// TIA Portal V17 export
// export: Created 2022-07-20T07:01:33.8166231Z, ExportSetting WithDefaults, DisplayName Totally Integrated Automation Portal, DisplayVersion V17, DisplayName TIA Portal Openness, DisplayVersion V17, DisplayName TIA Portal Version Control Interface, DisplayVersion V17, DisplayName SINAMICS Startdrive Advanced, DisplayVersion V17, DisplayName SINAMICS Startdrive G130, G150, S120, S150, SINAMICS MV, S210, DisplayVersion V17, DisplayName SINAMICS Startdrive G110M, G120, G120C, G120D, G120P, G115D, DisplayVersion V17, DisplayName STEP 7 Professional, DisplayVersion V17, DisplayName STEP 7 Safety, DisplayVersion V17, DisplayName WinCC Advanced, DisplayVersion V17
FUNCTION_BLOCK "FB10323_PrinterCompactAirCircuit"   // FB10323, LAD
{ S7_Optimized_Access := 'TRUE' }
VERSION : 0.1
// stored: AutoNumber false, IsIECCheckEnabled false, IsRetainMemResEnabled false, MemoryReserve 100, SetENOAutomatically false, UDAEnableTagReadback false
   VAR_INPUT
      AirCircuit_MainVacuum_VacuumSensor_raw : Int;
      AirCircuit_B1_VacuumSensor_raw : Int;
      AirCircuit_B2_VacuumSensor_raw : Int;
      AirCircuit_MainVacuum_Setpoint_mbar : Real;
      AirCircuit_B1_Setpoint_mbar : Real;
      AirCircuit_B2_Setpoint_mbar : Real;
      AirCircuitParameterB1PurgeTime_s : Time;
      AirCircuitParameterB2PurgeTime_s : Time;
   END_VAR
   VAR_OUTPUT
      AirCircuit_MainVacuum_SolenoidValve : Bool;
      AirCircuit_MainVacuum_Pump : Bool;
      AirCircuit_B1_JunctionMainVaccum_SolenoidValve : Bool;
      AirCircuit_B1_Tank_SolenoidValve : Bool;
      AirCircuit_B1_Venting_SolenoidValve : Bool;
      AirCircuit_B1_Purge_SolenoidValve : Bool;
      AirCircuit_B1_Purge_Pump : Bool;
      AirCircuit_B1_PurgeDone : Bool;
      AirCircuit_B2_JunctionMainVaccum_SolenoidValve : Bool;
      AirCircuit_B2_Tank_SolenoidValve : Bool;
      AirCircuit_B2_Venting_SolenoidValve : Bool;
      AirCircuit_B2_Purge_SolenoidValve : Bool;
      AirCircuit_B2_Purge_Pump : Bool;
      AirCircuit_B2_PurgeDone : Bool;
      EnablePWM : Bool;
      PumpDutyCycle : Int;
      MainVacuumActualValue : Real;
      B1VacuumActualValue : Real;
      AutoRegulationB1Done : Bool;
      B2VacuumActualValue : Real;
      AutoRegulationB2Done : Bool;
      AutoRegulationB1_B2_Done : Bool;
   END_VAR
   VAR_IN_OUT
      AirCircuitRequestAutoregulation : Bool;
      AirCircuitRequestMainVacuumRegulation : Bool;
      AirCircuitRequestB1Regulation : Bool;
      AirCircuitRequestB2Regulation : Bool;
      AirCircuitRequestB1Purge : Bool;
      AirCircuitRequestB2Purge : Bool;
   END_VAR
   VAR
      MainVacuumStateDiagram : Int;
      B1VacuumStateDiagram : Int;
      B2VacuumStateDiagram : Int;
      R_TRIG_RequestAutoregulationAirCircuit : R_TRIG;
      F_TRIG_RequestAutoregulationAirCircuit { S7_SetPoint := 'True'} : F_TRIG;
      R_TRIG_RequestMainVacuumRegulation { S7_SetPoint := 'True'} : R_TRIG;
      F_TRIG_RequestMainVacuumRegulation { S7_SetPoint := 'True'} : F_TRIG;
      R_TRIG_RequestB1Regulation { S7_SetPoint := 'True'} : R_TRIG;
      F_TRIG_RequestB1Regulation { S7_SetPoint := 'True'} : F_TRIG;
      R_TRIG_RequestB2Regulation { S7_SetPoint := 'True'} : R_TRIG;
      F_TRIG_RequestB2Regulation { S7_SetPoint := 'True'} : F_TRIG;
      R_TRIG_RequestB1Purge { S7_SetPoint := 'True'} : R_TRIG;
      R_TRIG_RequestB2Purge { S7_SetPoint := 'True'} : R_TRIG;
      FB10030_AnalogicalSensor_Instance { S7_SetPoint := 'True'} : "FB10030_AnalogicalSensor";
      MainVacuumCalibrationDataX1 { S7_SetPoint := 'True'} : Real;
      MainVacuumCalibrationDataY1 : Real;
      MainVacuumCalibrationDataX2 : Real;
      MainVacuumCalibrationDataY2 : Real;
      B1VacuumCalibrationDataX1 { S7_SetPoint := 'True'} : Real;
      B1VacuumCalibrationDataY1 : Real;
      B1VacuumCalibrationDataX2 : Real;
      B1VacuumCalibrationDataY2 : Real;
      B2VacuumCalibrationDataX1 : Real;
      B2VacuumCalibrationDataY1 : Real;
      B2VacuumCalibrationDataX2 : Real;
      B2VacuumCalibrationDataY2 : Real;
      TON_State11 { S7_SetPoint := 'True'} : TON_TIME;
      TON_State12 { S7_SetPoint := 'True'} : TON_TIME;
      TON_PurgeB1 { S7_SetPoint := 'True'} : TON_TIME;
      TON_PurgeB1_PumpEV_ON { S7_SetPoint := 'True'} : TON_TIME;
      TON_PurgeB1_PumpEV_OFF { S7_SetPoint := 'True'} : TON_TIME;
      TON_PurgeB1_EndOfPurge { S7_SetPoint := 'True'} : TON_TIME;
      TON_PurgeB2 { S7_SetPoint := 'True'} : TON_TIME;
      TON_PurgeB2_PumpEV_ON { S7_SetPoint := 'True'} : TON_TIME;
      TON_PurgeB2_PumpEV_OFF { S7_SetPoint := 'True'} : TON_TIME;
      TON_PurgeB2_EndOfPurge { S7_SetPoint := 'True'} : TON_TIME;
   END_VAR
   VAR CONSTANT
      "0_WAIT_FOR_AUTOREGULATION_REQUEST" : Int := 0;
      "10_MAINVACUUM_REGULATION" : Int := 10;
      "11_MAINVACUUM_PUMP_ACTIVATED" : Int := 11;
      "12_MAINVACUUM_PUMP_STOPPED" : Int := 12;
      "13_MAINVACCUM_REGULATED" : Int := 13;
      na : Int;
      "20_B1VACUUM_REGULATION" : Int := 20;
      "21_B1VACUUM_PUMP_ACTIVATED" : Int := 21;
      "22_B1VACUUM_REGULATED" : Int := 22;
      "25_B1PURGE_STATE1" : Int := 25;
      "26_B1PURGE_STATE2" : Int := 26;
      "27_B1PURGE_STATE3" : Int := 27;
      na_2 : Int;
      "30_B2VACUUM_REGULATION" : Int := 30;
      "31_B2VACUUM_PUMP_ACTIVATED" : Int := 31;
      "32_B2VACUUM_REGULATED" : Int := 32;
      "35_B2PURGE_STATE1" : Int := 35;
      "36_B2PURGE_STATE2" : Int := 36;
      "37_B2PURGE_STATE3" : Int := 37;
   END_VAR
BEGIN

REGION Network 1 (SCL): FirstScan
   IF "FirstScan" THEN
       #AirCircuit_MainVacuum_SolenoidValve := FALSE;
       #AirCircuit_MainVacuum_Pump := FALSE;
       #AirCircuit_B1_JunctionMainVaccum_SolenoidValve := FALSE;
       #AirCircuit_B1_Tank_SolenoidValve := FALSE;
       #AirCircuit_B1_Venting_SolenoidValve := FALSE;
       #AirCircuit_B1_Purge_SolenoidValve := FALSE;
       #AirCircuit_B2_JunctionMainVaccum_SolenoidValve := FALSE;
       #AirCircuit_B2_Tank_SolenoidValve := FALSE;
       #AirCircuit_B2_Venting_SolenoidValve := FALSE;
       #AirCircuit_B2_Purge_SolenoidValve := FALSE;

       #MainVacuumStateDiagram := #"10_MAINVACUUM_REGULATION";
       #B1VacuumStateDiagram := #"20_B1VACUUM_REGULATION";
       #B2VacuumStateDiagram := #"30_B2VACUUM_REGULATION";

       #PumpDutyCycle:= 100;
   END_IF;

   #MainVacuumCalibrationDataX1 := 0.0;
   #MainVacuumCalibrationDataY1 := 100.0;
   #MainVacuumCalibrationDataX2 := 27648.0;
   #MainVacuumCalibrationDataY2 := -100.0;

   #B1VacuumCalibrationDataX1 := 0.0;
   #B1VacuumCalibrationDataY1 := 100.0;
   #B1VacuumCalibrationDataX2 := 27648.0;
   #B1VacuumCalibrationDataY2 := -100.0;

   #B2VacuumCalibrationDataX1 := 0.0;
   #B2VacuumCalibrationDataY1 := 100.0;
   #B2VacuumCalibrationDataX2 := 27648.0;
   #B2VacuumCalibrationDataY2 := -100.0;
END_REGION

REGION Network 2 (SCL): EDGE SIGNAL AND TIMERS
   REGION EDGE SIGNAL
       #R_TRIG_RequestAutoregulationAirCircuit(CLK := #AirCircuitRequestAutoregulation);
       #F_TRIG_RequestAutoregulationAirCircuit(CLK := #AirCircuitRequestAutoregulation);

       #R_TRIG_RequestMainVacuumRegulation(CLK := #AirCircuitRequestMainVacuumRegulation);
       #F_TRIG_RequestMainVacuumRegulation(CLK := #AirCircuitRequestMainVacuumRegulation);

       #R_TRIG_RequestB1Regulation(CLK := #AirCircuitRequestB1Regulation);
       #F_TRIG_RequestB1Regulation(CLK := #AirCircuitRequestB1Regulation);

       #R_TRIG_RequestB2Regulation(CLK := #AirCircuitRequestB2Regulation);
       #F_TRIG_RequestB2Regulation(CLK := #AirCircuitRequestB2Regulation);

       #R_TRIG_RequestB1Purge(CLK := #AirCircuitRequestB1Purge);
       #R_TRIG_RequestB2Purge(CLK := #AirCircuitRequestB2Purge);
   END_REGION

   REGION TIMERS 
       #TON_State11(IN := #MainVacuumStateDiagram = #"11_MAINVACUUM_PUMP_ACTIVATED",
                    PT := T#100ms);
       #TON_State12(IN := #MainVacuumStateDiagram = #"12_MAINVACUUM_PUMP_STOPPED",
                    PT := T#100ms);

       #TON_PurgeB1(IN := (#B1VacuumStateDiagram = #"26_B1PURGE_STATE2") OR (#B1VacuumStateDiagram = #"25_B1PURGE_STATE1") ,
                    PT:= #AirCircuitParameterB1PurgeTime_s);

       #TON_PurgeB1_PumpEV_ON(IN := #B1VacuumStateDiagram = #"26_B1PURGE_STATE2" ,
                            PT := T#100ms);

       #TON_PurgeB1_PumpEV_OFF(IN := #B1VacuumStateDiagram = #"25_B1PURGE_STATE1" ,
                             PT := T#500ms);

       #TON_PurgeB1_EndOfPurge(IN := #B1VacuumStateDiagram = #"27_B1PURGE_STATE3",
                             PT := T#5s);

       #TON_PurgeB2(IN := (#B2VacuumStateDiagram = #"36_B2PURGE_STATE2") OR (#B2VacuumStateDiagram =#"35_B2PURGE_STATE1"),
                    PT := #AirCircuitParameterB2PurgeTime_s);

       #TON_PurgeB2_PumpEV_ON(IN := #B2VacuumStateDiagram = #"36_B2PURGE_STATE2",
                            PT := T#100ms);

     #TON_PurgeB2_PumpEV_OFF(IN := #B2VacuumStateDiagram = #"35_B2PURGE_STATE1",
                             PT := T#500ms);

     #TON_PurgeB2_EndOfPurge(IN := #B2VacuumStateDiagram = #"37_B2PURGE_STATE3",
                         PT := T#5s);

   END_REGION
END_REGION

REGION Network 3 (SCL): Air Circuit Statement Management
   #EnablePWM := #AirCircuitRequestAutoregulation OR #AirCircuitRequestMainVacuumRegulation OR #AirCircuitRequestB1Regulation OR #AirCircuitRequestB2Regulation;
END_REGION

REGION Network 4 (SCL): Air Circuit Management
   IF #R_TRIG_RequestAutoregulationAirCircuit.Q THEN
       #MainVacuumStateDiagram := #"11_MAINVACUUM_PUMP_ACTIVATED";
       #B1VacuumStateDiagram := #"21_B1VACUUM_PUMP_ACTIVATED";
       #B2VacuumStateDiagram := #"31_B2VACUUM_PUMP_ACTIVATED";
   END_IF;
   ////////////////////////////////////////////////////////////////////////////////::
   /////////////////////MAIN VACUUM
   CASE #MainVacuumStateDiagram OF

       #"10_MAINVACUUM_REGULATION":
           #AirCircuit_MainVacuum_SolenoidValve := FALSE;
           #AirCircuit_MainVacuum_Pump := FALSE;

           IF #R_TRIG_RequestMainVacuumRegulation.Q THEN
               #MainVacuumStateDiagram := #"11_MAINVACUUM_PUMP_ACTIVATED";
           END_IF;

       #"11_MAINVACUUM_PUMP_ACTIVATED":
           #AirCircuit_MainVacuum_SolenoidValve := FALSE;
           #AirCircuit_MainVacuum_Pump := TRUE;

           IF (#MainVacuumActualValue > #AirCircuit_MainVacuum_Setpoint_mbar) AND #TON_State11.Q THEN
               #MainVacuumStateDiagram := #"12_MAINVACUUM_PUMP_STOPPED";
           ELSIF (#MainVacuumActualValue <= #AirCircuit_MainVacuum_Setpoint_mbar) THEN
               #MainVacuumStateDiagram := #"13_MAINVACCUM_REGULATED";
           END_IF;

       #"12_MAINVACUUM_PUMP_STOPPED":
           #AirCircuit_MainVacuum_SolenoidValve := FALSE;
           #AirCircuit_MainVacuum_Pump := FALSE;

           IF (#MainVacuumActualValue > #AirCircuit_MainVacuum_Setpoint_mbar) AND #TON_State12.Q THEN
               #MainVacuumStateDiagram := #"11_MAINVACUUM_PUMP_ACTIVATED";
           ELSIF (#MainVacuumActualValue <= #AirCircuit_MainVacuum_Setpoint_mbar) THEN
               #MainVacuumStateDiagram := #"13_MAINVACCUM_REGULATED";
           END_IF;

       #"13_MAINVACCUM_REGULATED":
           #AirCircuit_MainVacuum_SolenoidValve := FALSE;
           #AirCircuit_MainVacuum_Pump := FALSE;

           IF (#MainVacuumActualValue > #AirCircuit_MainVacuum_Setpoint_mbar) THEN
               #MainVacuumStateDiagram := #"11_MAINVACUUM_PUMP_ACTIVATED";
           END_IF;

   END_CASE;

   ////////////////////////////////////////////////////////////////////////////////::
   /////////////////////B1 VACUUM
   CASE #B1VacuumStateDiagram OF

       #"20_B1VACUUM_REGULATION":
           #AirCircuit_B1_JunctionMainVaccum_SolenoidValve := FALSE;
           #AirCircuit_B1_Tank_SolenoidValve := FALSE;
           #AirCircuit_B1_Venting_SolenoidValve := FALSE;
           #AirCircuit_B1_Purge_SolenoidValve := FALSE;
           #AirCircuit_B1_Purge_Pump := FALSE;


           IF #R_TRIG_RequestB1Regulation.Q THEN
               #B1VacuumStateDiagram := #"21_B1VACUUM_PUMP_ACTIVATED";
           END_IF;

       #"21_B1VACUUM_PUMP_ACTIVATED":
           #AutoRegulationB1Done := FALSE;
           #AirCircuit_B1_JunctionMainVaccum_SolenoidValve := TRUE;
           #AirCircuit_B1_Tank_SolenoidValve := FALSE;
           #AirCircuit_B1_Venting_SolenoidValve := FALSE;
           #AirCircuit_B1_Purge_SolenoidValve := FALSE;
           #PumpDutyCycle := 100;
           IF (#B1VacuumActualValue <= #AirCircuit_B1_Setpoint_mbar) THEN
               #AutoRegulationB1Done := TRUE;
               #B1VacuumStateDiagram := #"22_B1VACUUM_REGULATED";
           END_IF;

       #"22_B1VACUUM_REGULATED":
           #AirCircuit_B1_JunctionMainVaccum_SolenoidValve := FALSE;
           #AirCircuit_B1_Tank_SolenoidValve := FALSE;
           #AirCircuit_B1_Venting_SolenoidValve := FALSE;
           #AirCircuit_B1_Purge_SolenoidValve := FALSE;

           IF (#B1VacuumActualValue > #AirCircuit_B1_Setpoint_mbar) THEN
               #B1VacuumStateDiagram := #"21_B1VACUUM_PUMP_ACTIVATED";
           ELSIF (#B1VacuumActualValue < #AirCircuit_B1_Setpoint_mbar - 0.5) THEN
               #AirCircuit_B1_JunctionMainVaccum_SolenoidValve := FALSE;
               #AirCircuit_B1_Tank_SolenoidValve := FALSE;
               #AirCircuit_B1_Venting_SolenoidValve := TRUE;
               #AirCircuit_B1_Purge_SolenoidValve := FALSE;
           END_IF;

       #"25_B1PURGE_STATE1":
           #AirCircuit_B1_JunctionMainVaccum_SolenoidValve := FALSE;
           #AirCircuit_B1_Tank_SolenoidValve := TRUE;
           #AirCircuit_B1_Venting_SolenoidValve := FALSE;
           #AirCircuit_B1_Purge_SolenoidValve := FALSE;
           #AirCircuit_B1_Purge_Pump := FALSE;
           #PumpDutyCycle := 50;

           IF #TON_PurgeB1_PumpEV_OFF.Q THEN
               #B1VacuumStateDiagram := #"26_B1PURGE_STATE2";
           END_IF;

       #"26_B1PURGE_STATE2":
           #AirCircuit_B1_JunctionMainVaccum_SolenoidValve := FALSE;
           #AirCircuit_B1_Tank_SolenoidValve := TRUE;
           #AirCircuit_B1_Venting_SolenoidValve := FALSE;
           #AirCircuit_B1_Purge_SolenoidValve := TRUE;
           #AirCircuit_B1_Purge_Pump := TRUE;

           IF #TON_PurgeB1_PumpEV_ON.Q THEN
               #B1VacuumStateDiagram := #"25_B1PURGE_STATE1";
           END_IF;

       #"27_B1PURGE_STATE3":
           #AirCircuit_B1_JunctionMainVaccum_SolenoidValve := FALSE;
           #AirCircuit_B1_Tank_SolenoidValve := TRUE;
           #AirCircuit_B1_Venting_SolenoidValve := FALSE;
           #AirCircuit_B1_Purge_SolenoidValve := FALSE;
           #AirCircuit_B1_Purge_Pump := FALSE;

           IF (#TON_PurgeB1_EndOfPurge.Q) THEN
               #AirCircuit_B1_PurgeDone := TRUE;
               #B1VacuumStateDiagram := #"21_B1VACUUM_PUMP_ACTIVATED";
           END_IF;

   END_CASE;

   IF (#TON_PurgeB1.Q) THEN
       #B1VacuumStateDiagram := #"27_B1PURGE_STATE3";
   END_IF;
   ////////////////////////////////////////////////////////////////////////////////::
   /////////////////////B2 VACUUM
   CASE #B2VacuumStateDiagram OF

       #"30_B2VACUUM_REGULATION":
           #AirCircuit_B2_JunctionMainVaccum_SolenoidValve := FALSE;
           #AirCircuit_B2_Tank_SolenoidValve := FALSE;
           #AirCircuit_B2_Venting_SolenoidValve := FALSE;
           #AirCircuit_B2_Purge_SolenoidValve := FALSE;
           #AirCircuit_B2_Purge_Pump := FALSE;

           IF #R_TRIG_RequestB2Regulation.Q THEN
               #B2VacuumStateDiagram := #"31_B2VACUUM_PUMP_ACTIVATED";
           END_IF;

       #"31_B2VACUUM_PUMP_ACTIVATED":
           #AutoRegulationB2Done := FALSE;
           #AirCircuit_B2_JunctionMainVaccum_SolenoidValve := TRUE;
           #AirCircuit_B2_Tank_SolenoidValve := FALSE;
           #AirCircuit_B2_Venting_SolenoidValve := FALSE;
           #AirCircuit_B2_Purge_SolenoidValve := FALSE;
           #PumpDutyCycle := 100;

           IF (#B2VacuumActualValue <= #AirCircuit_B2_Setpoint_mbar) THEN
               #AutoRegulationB2Done := TRUE;
               #B2VacuumStateDiagram := #"32_B2VACUUM_REGULATED";
           END_IF;

       #"32_B2VACUUM_REGULATED":
           #AirCircuit_B2_JunctionMainVaccum_SolenoidValve := FALSE;
           #AirCircuit_B2_Tank_SolenoidValve := FALSE;
           #AirCircuit_B2_Venting_SolenoidValve := FALSE;
           #AirCircuit_B2_Purge_SolenoidValve := FALSE;

           IF (#B2VacuumActualValue > #AirCircuit_B2_Setpoint_mbar) THEN
               #B2VacuumStateDiagram := #"31_B2VACUUM_PUMP_ACTIVATED";
           ELSIF (#B2VacuumActualValue < #AirCircuit_B2_Setpoint_mbar - 0.5) THEN
               #AirCircuit_B2_JunctionMainVaccum_SolenoidValve := FALSE;
               #AirCircuit_B2_Tank_SolenoidValve := FALSE;
               #AirCircuit_B2_Venting_SolenoidValve := TRUE;
               #AirCircuit_B2_Purge_SolenoidValve := FALSE;
           END_IF;


       #"35_B2PURGE_STATE1":
           #AirCircuit_B2_JunctionMainVaccum_SolenoidValve := FALSE;
           #AirCircuit_B2_Tank_SolenoidValve := TRUE;
           #AirCircuit_B2_Venting_SolenoidValve := FALSE;
           #AirCircuit_B2_Purge_SolenoidValve := FALSE;
           #AirCircuit_B2_Purge_Pump := FALSE;
           #PumpDutyCycle := 50;

           IF #TON_PurgeB2_PumpEV_OFF.Q THEN
               #B2VacuumStateDiagram := #"36_B2PURGE_STATE2";
           END_IF;

       #"36_B2PURGE_STATE2":
           #AirCircuit_B2_JunctionMainVaccum_SolenoidValve := FALSE;
           #AirCircuit_B2_Tank_SolenoidValve := TRUE;
           #AirCircuit_B2_Venting_SolenoidValve := FALSE;
           #AirCircuit_B2_Purge_SolenoidValve := TRUE;
           #AirCircuit_B2_Purge_Pump := TRUE;

           IF #TON_PurgeB2_PumpEV_ON.Q THEN
               #B2VacuumStateDiagram := #"35_B2PURGE_STATE1";
           END_IF;

       #"37_B2PURGE_STATE3":
           #AirCircuit_B2_JunctionMainVaccum_SolenoidValve := FALSE;
           #AirCircuit_B2_Tank_SolenoidValve := TRUE;
           #AirCircuit_B2_Venting_SolenoidValve := TRUE;
           #AirCircuit_B2_Purge_SolenoidValve := FALSE;
           #AirCircuit_B2_Purge_Pump := FALSE;

           IF (#TON_PurgeB2_EndOfPurge.Q) THEN
               #AirCircuit_B2_PurgeDone := TRUE;
               #B2VacuumStateDiagram := #"31_B2VACUUM_PUMP_ACTIVATED";
           END_IF;
   END_CASE;

   IF (#TON_PurgeB2.Q) THEN
       #B2VacuumStateDiagram := #"37_B2PURGE_STATE3";
   END_IF;

   ///////////////////////REQUEST////////////////////////
   IF #F_TRIG_RequestAutoregulationAirCircuit.Q  THEN
       #MainVacuumStateDiagram := #"10_MAINVACUUM_REGULATION";
       #B1VacuumStateDiagram := #"20_B1VACUUM_REGULATION";
       #B2VacuumStateDiagram := #"30_B2VACUUM_REGULATION";
   ELSIF #F_TRIG_RequestMainVacuumRegulation.Q  THEN
       #MainVacuumStateDiagram := #"10_MAINVACUUM_REGULATION";
   ELSIF #F_TRIG_RequestB1Regulation.Q THEN
       #B1VacuumStateDiagram := #"20_B1VACUUM_REGULATION";
   ELSIF #F_TRIG_RequestB2Regulation.Q THEN
       #B2VacuumStateDiagram := #"30_B2VACUUM_REGULATION";
   END_IF;


   /////////////////////////PURGE////////////////////////////
   //
   IF #R_TRIG_RequestB1Purge.Q THEN
       #AirCircuit_B1_PurgeDone := FALSE;
       #B1VacuumStateDiagram := #"25_B1PURGE_STATE1";
   END_IF;

   IF #R_TRIG_RequestB2Purge.Q THEN
       #AirCircuit_B2_PurgeDone := FALSE;
       #B2VacuumStateDiagram := #"35_B2PURGE_STATE1";
   END_IF;
END_REGION

REGION Network 5 (SCL): Air Circuit State Management
   #AutoRegulationB1_B2_Done := #AutoRegulationB1Done AND #AutoRegulationB2Done;
END_REGION

REGION Network 6
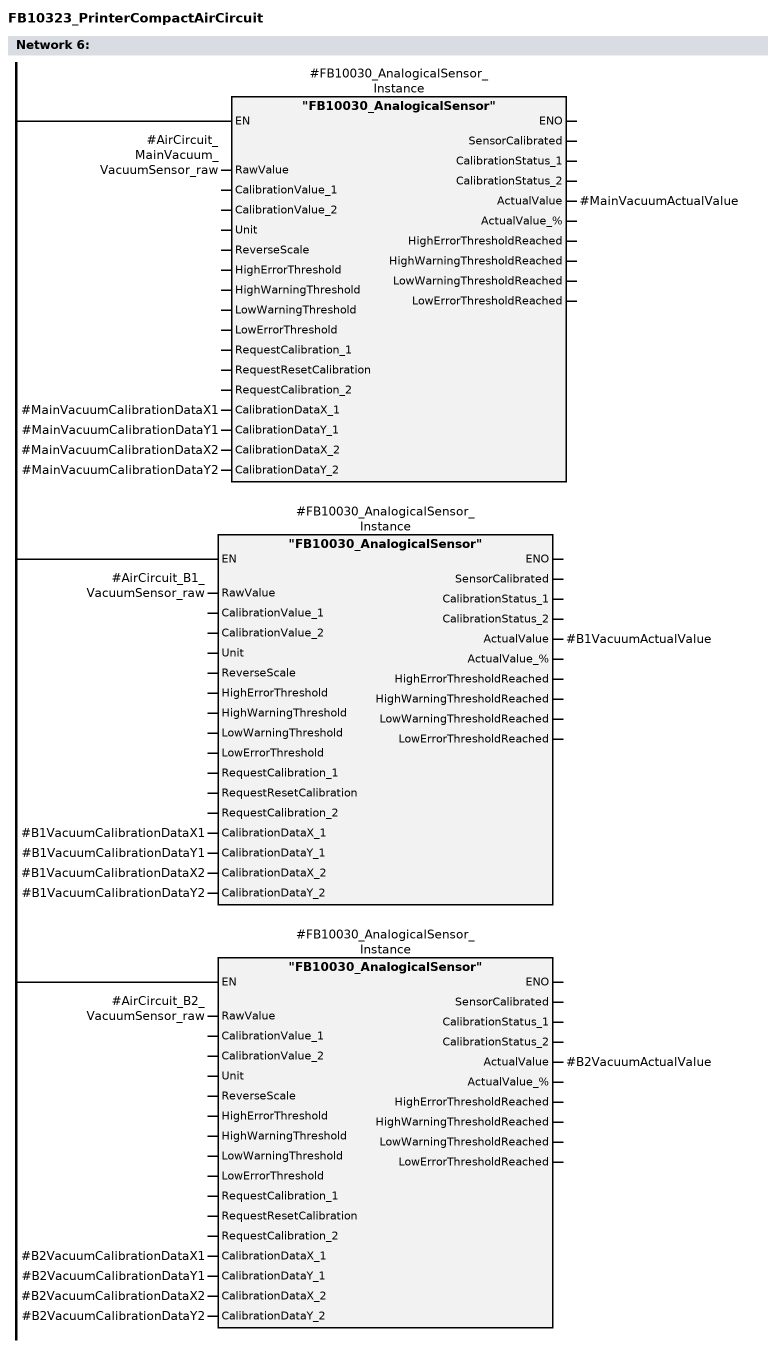
   RUNG wire#powerrail
      #FB10030_AnalogicalSensor_Instance(RawValue := #AirCircuit_MainVacuum_VacuumSensor_raw, CalibrationValue_1 :=, CalibrationValue_2 :=, Unit :=, HighErrorThreshold :=, HighWarningThreshold :=, LowWarningThreshold :=, LowErrorThreshold :=, RequestCalibration_1 :=, RequestCalibration_2 :=, RequestResetCalibration :=, CalibrationDataX_1 := #MainVacuumCalibrationDataX1, CalibrationDataY_1 := #MainVacuumCalibrationDataY1, CalibrationDataX_2 := #MainVacuumCalibrationDataX2, CalibrationDataY_2 := #MainVacuumCalibrationDataY2, SensorCalibrated =>, CalibrationStatus_1 =>, CalibrationStatus_2 =>, ActualValue => #MainVacuumActualValue, "ActualValue_%" =>, HighErrorThresholdReached =>, HighWarningThresholdReached =>, LowWarningThresholdReached =>, LowErrorThresholdReached =>, ReverseScale :=)
   END_RUNG
   RUNG wire#powerrail
      #FB10030_AnalogicalSensor_Instance(RawValue := #AirCircuit_B1_VacuumSensor_raw, CalibrationValue_1 :=, CalibrationValue_2 :=, Unit :=, HighErrorThreshold :=, HighWarningThreshold :=, LowWarningThreshold :=, LowErrorThreshold :=, RequestCalibration_1 :=, RequestCalibration_2 :=, RequestResetCalibration :=, CalibrationDataX_1 := #B1VacuumCalibrationDataX1, CalibrationDataY_1 := #B1VacuumCalibrationDataY1, CalibrationDataX_2 := #B1VacuumCalibrationDataX2, CalibrationDataY_2 := #B1VacuumCalibrationDataY2, SensorCalibrated =>, CalibrationStatus_1 =>, CalibrationStatus_2 =>, ActualValue => #B1VacuumActualValue, "ActualValue_%" =>, HighErrorThresholdReached =>, HighWarningThresholdReached =>, LowWarningThresholdReached =>, LowErrorThresholdReached =>, ReverseScale :=)
   END_RUNG
   RUNG wire#powerrail
      #FB10030_AnalogicalSensor_Instance(RawValue := #AirCircuit_B2_VacuumSensor_raw, CalibrationValue_1 :=, CalibrationValue_2 :=, Unit :=, HighErrorThreshold :=, HighWarningThreshold :=, LowWarningThreshold :=, LowErrorThreshold :=, RequestCalibration_1 :=, RequestCalibration_2 :=, RequestResetCalibration :=, CalibrationDataX_1 := #B2VacuumCalibrationDataX1, CalibrationDataY_1 := #B2VacuumCalibrationDataY1, CalibrationDataX_2 := #B2VacuumCalibrationDataX2, CalibrationDataY_2 := #B2VacuumCalibrationDataY2, SensorCalibrated =>, CalibrationStatus_1 =>, CalibrationStatus_2 =>, ActualValue => #B2VacuumActualValue, "ActualValue_%" =>, HighErrorThresholdReached =>, HighWarningThresholdReached =>, LowWarningThresholdReached =>, LowErrorThresholdReached =>, ReverseScale :=)
   END_RUNG
   // the same network as SCL:
   #FB10030_AnalogicalSensor_Instance(RawValue := #AirCircuit_MainVacuum_VacuumSensor_raw,   // "FB10030_AnalogicalSensor"
                           CalibrationDataX_1 := #MainVacuumCalibrationDataX1,
                           CalibrationDataY_1 := #MainVacuumCalibrationDataY1,
                           CalibrationDataX_2 := #MainVacuumCalibrationDataX2,
                           CalibrationDataY_2 := #MainVacuumCalibrationDataY2,
                           ActualValue => #MainVacuumActualValue);
   #FB10030_AnalogicalSensor_Instance(RawValue := #AirCircuit_B1_VacuumSensor_raw,   // "FB10030_AnalogicalSensor"
                           CalibrationDataX_1 := #B1VacuumCalibrationDataX1,
                           CalibrationDataY_1 := #B1VacuumCalibrationDataY1,
                           CalibrationDataX_2 := #B1VacuumCalibrationDataX2,
                           CalibrationDataY_2 := #B1VacuumCalibrationDataY2,
                           ActualValue => #B1VacuumActualValue);
   #FB10030_AnalogicalSensor_Instance(RawValue := #AirCircuit_B2_VacuumSensor_raw,   // "FB10030_AnalogicalSensor"
                           CalibrationDataX_1 := #B2VacuumCalibrationDataX1,
                           CalibrationDataY_1 := #B2VacuumCalibrationDataY1,
                           CalibrationDataX_2 := #B2VacuumCalibrationDataX2,
                           CalibrationDataY_2 := #B2VacuumCalibrationDataY2,
                           ActualValue => #B2VacuumActualValue);
END_REGION
END_FUNCTION_BLOCK
